(* Logix 5000 project; controller AMANA_DC_ASSEMBLY_01 vendor 1 type 14 code 166 rev 31.11; software revision 31.02 *)

TASK MainTask (continuous, watchdog 500 ms) : MainProgram

MODULES
   Local : vendor 1 type 14 code 166 (ICP 0, rev 31.11)
END_MODULES

PROGRAM MainProgram   (* main routine MainRoutine *)

ROUTINE MainRoutine   (* ladder *)
END_ROUTINE
END_PROGRAM
